INTERFACE I_ObjectRunner

METHOD DeregisterAllModules : HRESULT
VAR_INPUT
END_VAR
END_METHOD

METHOD RegisterModule : HRESULT
VAR_INPUT
	CyclicModule : ICyclic;
END_VAR
END_METHOD

END_INTERFACE

(* stored: Version 1.1.0.1
   Itf I_ObjectRunner: Id {7ae64750-6a2f-446f-b3b5-fa2d9501c423}
   Method DeregisterAllModules: Id {cd468435-7f31-474e-b797-49d6e54c3deb}
   Method RegisterModule: Id {119d0526-b150-47f1-ab98-856e052618fb} *)
